INTERFACE I_ValidateInterface EXTENDS I_Debug

{attribute 'hide'}
METHOD ValidateInterface
VAR_INPUT
END_VAR
END_METHOD

END_INTERFACE

(* stored: Version 1.1.0.1
   Itf I_ValidateInterface: Id {437a69c8-a4e0-4a55-a63e-9368065bdc44}
   Method ValidateInterface: Id {540c56c6-6fcf-44ac-8e48-d827e929ffe3} *)
